(* IEC 61131-3 sources: stc/cmd/stc-mcp/testdata/live, 4 files *)

(* ---- types.st ---- *)
TYPE ST_Conveyor_HMI :
STRUCT
	p_cmd_Start : BOOL;
	p_cmd_Stop : BOOL;
	p_stat_Running : BOOL;
	p_stat_Sensor : BOOL;
	p_cfg_Speed : INT := 50;
END_STRUCT
END_TYPE

(* ---- GVL_Live.st ---- *)
// Live session fixture for the stc-mcp sim tools: one conveyor with an HMI
// struct, a sensor input linked to Demo Device 1's EL1008 channel 1 and a
// running-cycle counter.
{attribute 'qualified_only'}
VAR_GLOBAL
	{attribute 'OPC.UA.DA' := '1'}
	conveyor : FB_Conveyor;
	{attribute 'TcLinkTo' := 'TIID^Device 1 (EtherCAT)^DEMO.A1.00 (EK1200)^DEMO.A1.01 (EL1008)^Channel 1^Input'}
	{attribute 'OPC.UA.DA' := '1'}
	xSensor AT %I* : BOOL;
	{attribute 'OPC.UA.DA' := '1'}
	nRunCycles : DINT;
END_VAR
VAR_GLOBAL CONSTANT
	cMax : INT := 10;
END_VAR

(* ---- fbs.st ---- *)
FUNCTION_BLOCK FB_Conveyor
VAR_INPUT
	xSensor : BOOL;
END_VAR
VAR_OUTPUT
	xRunning : BOOL;
END_VAR
VAR
	{attribute 'OPC.UA.DA' := '1'}
	HMI : ST_Conveyor_HMI;
END_VAR
IF HMI.p_cmd_Start THEN
	HMI.p_stat_Running := TRUE;
	HMI.p_cmd_Start := FALSE;
END_IF;
IF HMI.p_cmd_Stop THEN
	HMI.p_stat_Running := FALSE;
	HMI.p_cmd_Stop := FALSE;
END_IF;
HMI.p_stat_Sensor := xSensor;
xRunning := HMI.p_stat_Running;
END_FUNCTION_BLOCK

(* ---- main.st ---- *)
PROGRAM MAIN
GVL_Live.conveyor(xSensor := GVL_Live.xSensor);
IF GVL_Live.conveyor.xRunning THEN
	GVL_Live.nRunCycles := GVL_Live.nRunCycles + 1;
END_IF;
END_PROGRAM
